FUNCTION_BLOCK SS3_ifb_ps_Camera (* Composite FB wrapping other FBs *)
  (* Standard: 61499-2 *)
  (* Version 1.0, 2025-05-26, PS_Transformer_for_Unknown *)
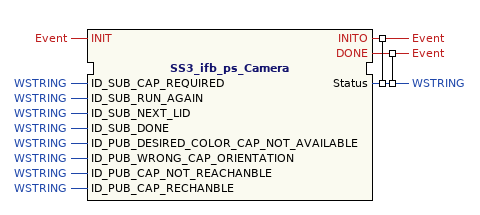
  EVENT_INPUT
    INIT; (* Initialization Request *)
  END_EVENT
  EVENT_OUTPUT
    INITO WITH Status; (* Initialization Confirm *)
    DONE WITH Status; (* Execution Confirmation *)
  END_EVENT
  VAR_INPUT
    ID_SUB_CAP_REQUIRED : WSTRING;
    ID_SUB_RUN_AGAIN : WSTRING;
    ID_SUB_NEXT_LID : WSTRING;
    ID_SUB_DONE : WSTRING;
    ID_PUB_DESIRED_COLOR_CAP_NOT_AVAILABLE : WSTRING;
    ID_PUB_WRONG_CAP_ORIENTATION : WSTRING;
    ID_PUB_CAP_NOT_REACHANBLE : WSTRING;
    ID_PUB_CAP_RECHANBLE : WSTRING;
  END_VAR
  VAR_OUTPUT
    Status : WSTRING; (* Output event qualifier *)
  END_VAR
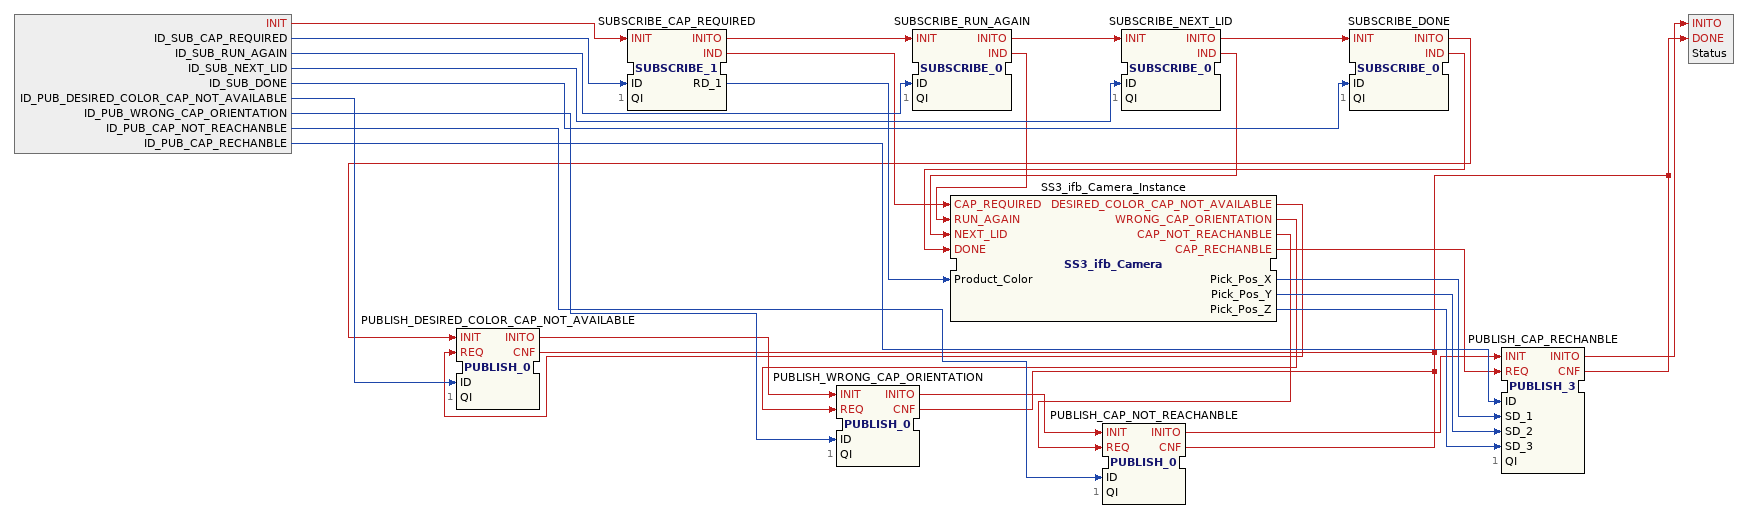
  FBS
    SS3_ifb_Camera_Instance : SS3_ifb_Camera;
    SUBSCRIBE_CAP_REQUIRED : SUBSCRIBE_1(QI := 1);
    SUBSCRIBE_RUN_AGAIN : SUBSCRIBE_0(QI := 1);
    SUBSCRIBE_NEXT_LID : SUBSCRIBE_0(QI := 1);
    SUBSCRIBE_DONE : SUBSCRIBE_0(QI := 1);
    PUBLISH_DESIRED_COLOR_CAP_NOT_AVAILABLE : PUBLISH_0(QI := 1);
    PUBLISH_WRONG_CAP_ORIENTATION : PUBLISH_0(QI := 1);
    PUBLISH_CAP_NOT_REACHANBLE : PUBLISH_0(QI := 1);
    PUBLISH_CAP_RECHANBLE : PUBLISH_3(QI := 1);
  END_FBS
  EVENT_CONNECTIONS
    INIT TO SUBSCRIBE_CAP_REQUIRED.INIT;
    SUBSCRIBE_CAP_REQUIRED.INITO TO SUBSCRIBE_RUN_AGAIN.INIT;
    SUBSCRIBE_RUN_AGAIN.INITO TO SUBSCRIBE_NEXT_LID.INIT;
    SUBSCRIBE_NEXT_LID.INITO TO SUBSCRIBE_DONE.INIT;
    SUBSCRIBE_DONE.INITO TO PUBLISH_DESIRED_COLOR_CAP_NOT_AVAILABLE.INIT;
    PUBLISH_DESIRED_COLOR_CAP_NOT_AVAILABLE.INITO TO PUBLISH_WRONG_CAP_ORIENTATION.INIT;
    PUBLISH_WRONG_CAP_ORIENTATION.INITO TO PUBLISH_CAP_NOT_REACHANBLE.INIT;
    PUBLISH_CAP_NOT_REACHANBLE.INITO TO PUBLISH_CAP_RECHANBLE.INIT;
    PUBLISH_CAP_RECHANBLE.INITO TO INITO;
    SUBSCRIBE_CAP_REQUIRED.IND TO SS3_ifb_Camera_Instance.CAP_REQUIRED;
    SUBSCRIBE_RUN_AGAIN.IND TO SS3_ifb_Camera_Instance.RUN_AGAIN;
    SUBSCRIBE_NEXT_LID.IND TO SS3_ifb_Camera_Instance.NEXT_LID;
    SUBSCRIBE_DONE.IND TO SS3_ifb_Camera_Instance.DONE;
    SS3_ifb_Camera_Instance.DESIRED_COLOR_CAP_NOT_AVAILABLE TO PUBLISH_DESIRED_COLOR_CAP_NOT_AVAILABLE.REQ;
    SS3_ifb_Camera_Instance.WRONG_CAP_ORIENTATION TO PUBLISH_WRONG_CAP_ORIENTATION.REQ;
    SS3_ifb_Camera_Instance.CAP_NOT_REACHANBLE TO PUBLISH_CAP_NOT_REACHANBLE.REQ;
    SS3_ifb_Camera_Instance.CAP_RECHANBLE TO PUBLISH_CAP_RECHANBLE.REQ;
    PUBLISH_DESIRED_COLOR_CAP_NOT_AVAILABLE.CNF TO DONE;
    PUBLISH_WRONG_CAP_ORIENTATION.CNF TO DONE;
    PUBLISH_CAP_NOT_REACHANBLE.CNF TO DONE;
    PUBLISH_CAP_RECHANBLE.CNF TO DONE;
  END_CONNECTIONS
  DATA_CONNECTIONS
    ID_SUB_CAP_REQUIRED TO SUBSCRIBE_CAP_REQUIRED.ID;
    ID_SUB_RUN_AGAIN TO SUBSCRIBE_RUN_AGAIN.ID;
    ID_SUB_NEXT_LID TO SUBSCRIBE_NEXT_LID.ID;
    ID_SUB_DONE TO SUBSCRIBE_DONE.ID;
    ID_PUB_DESIRED_COLOR_CAP_NOT_AVAILABLE TO PUBLISH_DESIRED_COLOR_CAP_NOT_AVAILABLE.ID;
    ID_PUB_WRONG_CAP_ORIENTATION TO PUBLISH_WRONG_CAP_ORIENTATION.ID;
    ID_PUB_CAP_NOT_REACHANBLE TO PUBLISH_CAP_NOT_REACHANBLE.ID;
    ID_PUB_CAP_RECHANBLE TO PUBLISH_CAP_RECHANBLE.ID;
    SUBSCRIBE_CAP_REQUIRED.RD_1 TO SS3_ifb_Camera_Instance.Product_Color;
    SS3_ifb_Camera_Instance.Pick_Pos_X TO PUBLISH_CAP_RECHANBLE.SD_1;
    SS3_ifb_Camera_Instance.Pick_Pos_Y TO PUBLISH_CAP_RECHANBLE.SD_2;
    SS3_ifb_Camera_Instance.Pick_Pos_Z TO PUBLISH_CAP_RECHANBLE.SD_3;
  END_CONNECTIONS
END_FUNCTION_BLOCK
